// TIA Portal V16 export
// export: Created 2024-12-03T15:41:44.9072209Z, ExportSetting WithReadOnly, DisplayName Totally Integrated Automation Portal, DisplayVersion V16 Update 6, DisplayName TIA Portal Version Control Interface, DisplayVersion V16 Update 2, DisplayName TIA Portal Openness, DisplayVersion V16 Update 6, DisplayName TIA Portal Teamcenter Gateway, DisplayVersion V16, DisplayName SINAMICS Startdrive Advanced, DisplayVersion V16 Update 5, DisplayName SINAMICS Startdrive G130, G150, S120, S150, SINAMICS MV, S210, DisplayVersion V16 Update 5, DisplayName SINAMICS Startdrive G110M, G120, G120C, G120D, G120P, G115D, DisplayVersion V16 Update 5, DisplayName STEP 7 Professional, DisplayVersion V16 Update 6, DisplayName STEP 7 Safety, DisplayVersion V16, DisplayName WinCC Advanced / Unified PC, DisplayVersion V16 Update 6
TYPE "CLXAiPLC_IN_UDT"
// stored: CreationDate 2021-07-13T07:41:36.2278727Z, InterfaceModifiedDate 2019-12-05T06:59:16.4729649Z, IsConsistent true, LibraryConformanceStatus The object is library-conformant., ModifiedDate 2021-03-27T07:36:50.6243175Z
   STRUCT
      Convey_stop_status { ExternalVisible := 'False'} : Struct   // Status of ConveyStop
         Reserved0 : Bool;
         Reserved1 : Bool;
         StopActiveCommandPLC : Bool;   // Stop active due to stop command from the PLC
         Reserved3 : Bool;
         Reserved4 : Bool;
         Reserved5 : Bool;
         Reserved6 : Bool;
         Reserved7 : Bool;
         Reserved8 : Bool;
         Reserved9 : Bool;
         Reserved10 : Bool;
         Reserved11 : Bool;
         Reserved12 : Bool;
         StopActiveOtherModule : Bool;   // Stop condition is active on a module in the ConveyStop group
         StopActiveLostConn : Bool;   // Stop is active due to a loss of communication connection
         StopActiveLostPLC : Bool;   // Stop active due to a loss of connection with the PLC
      END_STRUCT;
      AllSensors { ExternalVisible := 'False'} : Struct   // All sensor inputs
         "Reserved[0]" : Bool;
         "Reserved[1]" : Bool;
         "Reserved[2]" : Bool;
         "Reserved[3]" : Bool;
         "Reserved[4]" : Bool;
         "Reserved[5]" : Bool;
         "Reserved[6]" : Bool;
         Heartbeat : Bool;   // This bit toggles every 2 seconds .
         LeftPin2 : Bool;   // Left sensor port state (Pin2)
         "Reserved[9]" : Bool;
         RightPin2 : Bool;   // Right sensor port state (Pin2)
         "Reserved[11]" : Bool;
         LeftPin4 : Bool;   // Left sensor port state (Pin4)
         "Reserved[13]" : Bool;
         RightPin4 : Bool;   // Right sensor port state (Pin4)
         "Reserved[15]" : Bool;
      END_STRUCT;
      SensorDetect { ExternalVisible := 'False'} : Struct   // Sensor detection
         Reserved : Byte;
         RightSensorDetect : Bool;   // If this bit is TRUE a sensor has been detected on the Right sensor port
         LeftSensorDetect : Bool;   // If this bit is TRUE a sensor has been detected on the Left sensor port
         "Reserved[10]" : Bool;
         "Reserved[11]" : Bool;
         "Reserved[12]" : Bool;
         "Reserved[13]" : Bool;
         "Reserved[14]" : Bool;
         "Reserved[15]" : Bool;
      END_STRUCT;
      Voltage { ExternalVisible := 'False'} : Int;   // The Voltage applied to the module in milivolts
      LeftCurrent { ExternalVisible := 'False'} : Int;   // The current consumed by the Left MDR in miliamperes
      LeftFreq { ExternalVisible := 'False'} : Int;   // MDR frequency in Hz as measured by the Hall effect sensors
      LeftCalcTemp { ExternalVisible := 'False'} : Byte;   // The temperature of the Left MDR in degrees Celsius
      ModuleTemp { ExternalVisible := 'False'} : Byte;   // The temperature of the module in degrees Celsius
      LeftMDRDiagnostic { ExternalVisible := 'False'} : Struct   // Left MDR diagnostics .
         Overheat : Bool;   // The MDR 's temperature has exceeded 105 degrees Celsius
         MaxTorque : Bool;   // The MDR is running with maximum torque output
         ShortCircuit : Bool;   // There is a short circuit on the MDR
         MDRNotConnected : Bool;   // The MDR is not connected
         Overload : Bool;   // The MDR has been overloaded - this means its speed is less than 10% of the selected speed
         Stalled : Bool;   // The MDR has stalled
         MDRBadHall : Bool;   // The MDR has a Hall Efect Sensor error
         MDRNotUsed : Bool;   // The MDR is not used
         MDRStatus1 : Bool;   // This field and the next are used together by the module to indicate the status of the MDR. Please refer to documentation
         MDRStatus2 : Bool;
         MDRinDOmode : Bool;   // The MDR is in digital Output mode .
         Reserved1 : Bool;
         Reserved2 : Bool;
         Reserved3 : Bool;
         OverVoltage : Bool;   // The sum of the module power supply voltage + the MDR-generated voltage has exceeded 30 volts
         LowVoltage : Bool;   // Module power supply is less than 18 Volts
      END_STRUCT;
      RightCurrent { ExternalVisible := 'False'} : Int;   // The current consumed by the Right motor in miliamperes
      RightFreq { ExternalVisible := 'False'} : Int;   // MDR frequency in Hz as measured by the Hall effect sensors
      RightCalcTemp { ExternalVisible := 'False'} : Byte;   // The temperature of the Right MDR in degrees Celsius
      ModuleTemp_1 { ExternalVisible := 'False'} : Byte;   // The temperature of the module in degrees Celsius
      RightMDRDiagnostic { ExternalVisible := 'False'} : Struct   // Right MDR diagnostics .
         Overheat : Bool;   // The MDR 's temperature has exceeded 105 degrees Celsius
         MaxTorque : Bool;   // The MDR is running with maximum torque output
         ShortCircuit : Bool;   // There is a short circuit on the MDR
         MDRNotConnected : Bool;   // The MDR is not connected
         Overload : Bool;   // The MDR has been overloaded - this means its speed is less than 10% of the selected speed
         Stalled : Bool;   // The MDR has stalled
         MDRBadHall : Bool;   // The MDR has a Hall Efect Sensor error
         MDRNotUsed : Bool;   // The MDR is not used
         MDRStatus1 : Bool;   // This field and the next are used together by the module to indicate the status of the MDR. Please refer to documentation
         MDRStatus2 : Bool;
         MDRinDOmode : Bool;   // The MDR is in digital Output mode .
         Reserved1 : Bool;
         Reserved2 : Bool;
         Reserved3 : Bool;
         OverVoltage : Bool;   // The sum of the module power supply voltage + the MDR-generated voltage has exceeded 30 volts
         LowVoltage : Bool;   // Module power supply is less than 18 Volts
      END_STRUCT;
      LeftMDR_DIOstatus : Struct   // This is the status when the MDR is used as a digital IO
         Reserved0 : Bool;
         Reserved1 : Bool;
         Reserved2 : Bool;
         Reserved3 : Bool;
         ShortCircuit : Bool;   // When this bit is '1' , there is a short circuit between +24V and Pin2/3/4
         Reserved5 : Bool;
         Reserved6 : Bool;
         Reserved7 : Bool;
         Reserved : Byte;
      END_STRUCT;
      RightMDR_DIOstatus : Struct   // This is the status when the MDR is used as a digital IO
         Reserved0 : Bool;
         Reserved1 : Bool;
         Reserved2 : Bool;
         Reserved3 : Bool;
         ShortCircuit : Bool;   // When this bit is '1' , there is a short circuit between +24V and Pin2/3/4
         Reserved5 : Bool;
         Reserved6 : Bool;
         Reserved7 : Bool;
         Reserved : Byte;
      END_STRUCT;
      UpstreamModuleStatus { ExternalVisible := 'False'} : Word;   // The ZPA status from the Upstream ConveyLinx module
      DownstreamModuleStatus { ExternalVisible := 'False'} : Word;   // The ZPA status from the Downstream ConveyLinx module
      TrackingFromUpstream { ExternalVisible := 'False'} : DWord;   // Tracking data from the Upstream ConveyLinx module
      Reserved { ExternalVisible := 'False'} : Word;
      DistanceLeft { ExternalVisible := 'False'} : Int;   // Distance traveled by the Left MDR in 'mm'. For all Servo commands and statuses , please refer to documentation
      DistanceRight { ExternalVisible := 'False'} : Int;   // Distance traveled by the Right MDR in 'mm'
      ServoStatusLeft { ExternalVisible := 'False'} : Struct   // Status Word for Servo commands for Left MDR
         Reserve_6 : Byte;
         LastServoCommandExecuted : Bool;
         ResetPulseCount_Echo : Bool;
         RunCommand_Echo : Bool;
         Reserve_1 : Bool;
         Reserve_2 : Bool;
         Reserve_3 : Bool;
         Reserve_4 : Bool;
         Reserve_5 : Bool;
      END_STRUCT;
      ServoStatusRight { ExternalVisible := 'False'} : Struct   // Status Word for Servo commands for Right MDR
         Reserve_6 : Byte;
         LastServoCommandExecuted : Bool;
         ResetPulseCount_Echo : Bool;
         RunCommand_Echo : Bool;
         Reserve_1 : Bool;
         Reserve_2 : Bool;
         Reserve_3 : Bool;
         Reserve_4 : Bool;
         Reserve_5 : Bool;
      END_STRUCT;
      LeftMDRRealSpeed { ExternalVisible := 'False'} : Word;   // The Real Speed of the MDR in m/sec*1000 . Also two status bits are included . Please refer to documentation
      RightMDRRealSpeed { ExternalVisible := 'False'} : Word;   // The Real Speed of the MDR in m/sec*1000 . Also two status bits are included . Please refer to documentation
      Future { ExternalVisible := 'False'} : Array[25..31] of Word;
   END_STRUCT;
END_TYPE
